# EPICS autosave request: GALILMUL/iocBoot/iocGALILMUL-IOC-01/GALILMUL_01_positions_norestore.req
# we keep a copy of current positions, but this file is not specified
# as part of an autosave load at boot time
file "GALIL_controller_positions.req" "P=$(P),CCP=$(MTRCTRL1)"
file "GALIL_controller_positions.req" "P=$(P),CCP=$(MTRCTRL2)"
